TYPE E_LATState :
(
	eLAT_Stop :=0,
	eLAT_Startup:=1,
	eLAT_Ready:=2,
	eLAT_InOperation:=3,
	eLAT_Passive:=4
);
END_TYPE

(* stored: Version 1.1.0.1, ProductVersion 3.1.4024.9
   DUT E_LATState: Id {94fe921f-33f9-4063-b70e-f0593a12ae76} *)
